INTERFACE I_GraphFramework

METHOD PUBLIC Create : I_Graph
VAR_INPUT
END_VAR
END_METHOD

PROPERTY PUBLIC Datatypes : I_Datatypes
GET
END_GET
END_PROPERTY

METHOD PUBLIC Install
VAR_INPUT
	Pack : I_GraphPack;
END_VAR
END_METHOD

PROPERTY PUBLIC NodeFactory : I_NodeFactory
GET
END_GET
END_PROPERTY

END_INTERFACE

(* stored: Version 1.1.0.1, ProductVersion 3.1.4024.12
   Itf I_GraphFramework: Id {f3353d67-fe68-422a-8558-089dff4b9a79}
   Method Create: Id {ac947962-8060-47be-8a13-b27b6702168a}
   Property Datatypes: Id {aaf13d06-2670-4934-aa21-f9395287f1c7}
   Get Get: Id {71680b95-9334-4f3e-9564-42b2ba265567}
   Method Install: Id {1b3dea12-ac6d-0c7a-30a8-f1233e671c1b}
   Property NodeFactory: Id {edf7f767-4697-41c5-b9ba-9bf9e9d25a3b}
   Get Get: Id {f1017b5c-4b53-42cc-8ed6-f8ae79e6a313} *)
